(* PLC project Unnamed, Unknown Unnamed 1 *)
(* stored: creationDateTime 2024-11-02T19:05:21, modificationDateTime 2024-11-03T20:00:09 *)

PROGRAM WaterTank
  VAR CONSTANT
    max_level AT %QW1 : INT := 100;
  END_VAR
  VAR CONSTANT
    true0 : BOOL := 1;
    false0 : BOOL := 0;
    three : INT := 2;
    zero : INT := 0;
  END_VAR
  VAR CONSTANT
    min_level AT %QW2 : INT := 0;
  END_VAR
  VAR
    pump_speed AT %QW3 : INT := 0;
    pump_state AT %QX0.0 : BOOL;
    pump_control AT %QX0.1 : BOOL := 0;
    man_button AT %QX0.3 : BOOL := 1;
    manual_control AT %QX0.2 : BOOL := 0;
    water_level AT %IW0 : INT := 50;
    rising_level AT %QW4 : INT := 1;
  END_VAR
  VAR  (* added by the conversion: wires and edge detectors of the diagram *)
    _MOVE50_ENO : BOOL;
    _MOVE50_OUT : INT;
    _GE31_ENO : BOOL;
    _GE31_OUT : BOOL;
    _LT69_ENO : BOOL;
    _LT69_OUT : BOOL;
    _GT71_ENO : BOOL;
    _GT71_OUT : BOOL;
  END_VAR

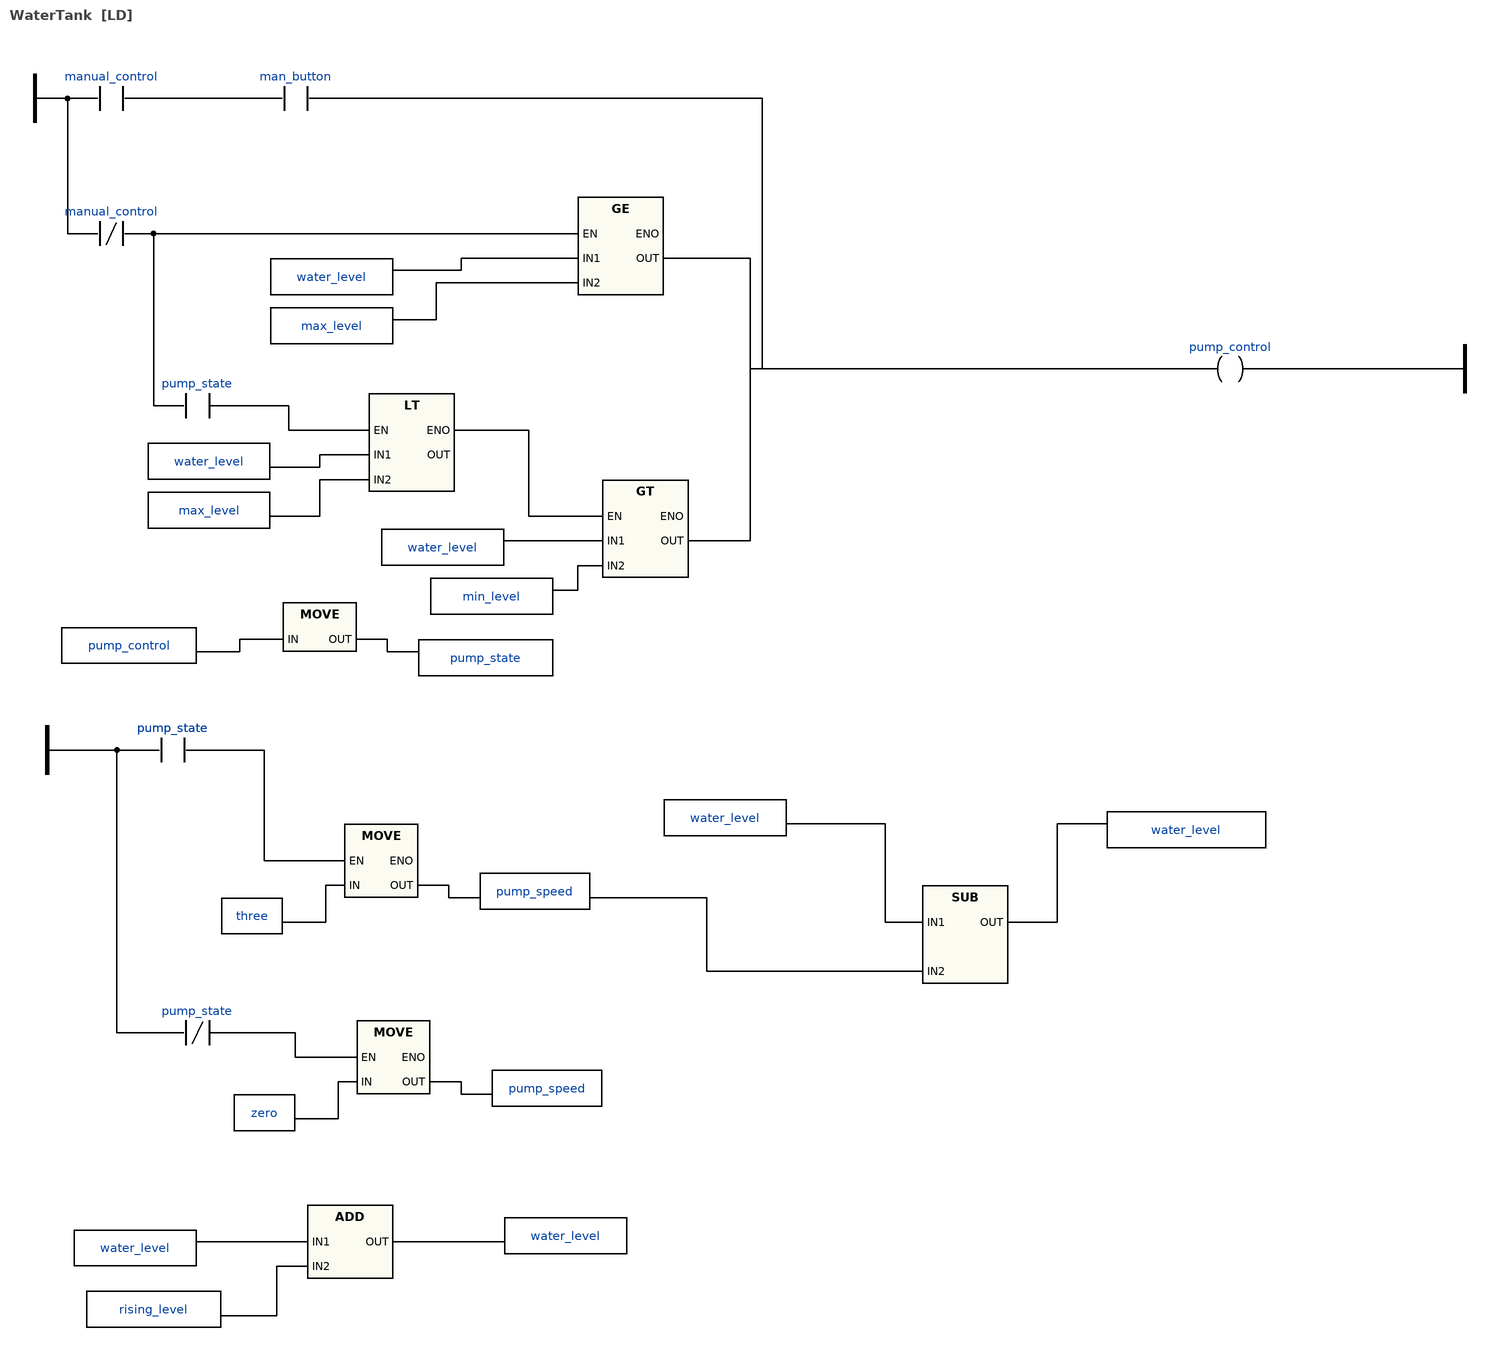
(* LD diagram, written out as Structured Text *)
water_level := water_level - pump_speed;
water_level := water_level + rising_level;
_MOVE50_OUT := MOVE(EN := pump_state, IN := three, ENO => _MOVE50_ENO);
IF _MOVE50_ENO THEN pump_speed := _MOVE50_OUT; END_IF;
IF NOT pump_state THEN pump_speed := zero; END_IF;
_GE31_OUT := GE(EN := NOT manual_control, IN1 := water_level, IN2 := max_level, ENO => _GE31_ENO);
_LT69_OUT := LT(EN := NOT manual_control AND pump_state, IN1 := water_level, IN2 := max_level, ENO => _LT69_ENO);
_GT71_OUT := GT(EN := _LT69_ENO, IN1 := water_level, IN2 := min_level, ENO => _GT71_ENO);
pump_control := _GE31_OUT OR _GT71_OUT OR manual_control AND man_button;
pump_state := pump_control;
(* drawn but not wired to any output: pump_state *)
END_PROGRAM

CONFIGURATION Config0
  RESOURCE Res0 ON PLC
    TASK task0(INTERVAL := T#20ms, PRIORITY := 0);
    PROGRAM instance0 WITH task0 : WaterTank;
  END_RESOURCE
END_CONFIGURATION
